(* CODESYS project EX1.project

Project tree, tasks and I/O mapping:
  Device : CODESYS Control Win V3, 3S - Smart Software Solutions GmbH, order no. 305021, version 3.5.11.30
    application Application
      libraries: Standard, * (System)
      task MainTask (cyclic, interval t#20ms, priority 1) calls PLC_PRG
      program PLC_PRG [LD]
*)

// Device/Application/PLC_PRG
PROGRAM PLC_PRG
VAR
	B1 : BOOL;     // BOTOEIRA DE ENTRADA B1
	B2 : BOOL;     // BOTOEIRA DE ENTRADA B2
	K1 : BOOL;     // MOTOR
END_VAR

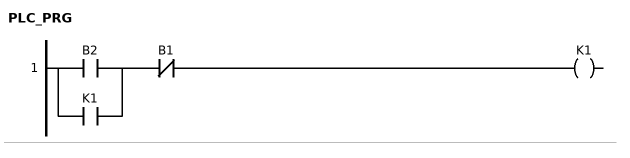
// NETWORK 1
K1 := (B2 OR K1) AND NOT B1;

END_PROGRAM
